// TwinCAT 3 PLC project FTP
// ProgramVersion: 3.1.4023.0
// libraries:
//   Tc2_FTP, * (Beckhoff Automation GmbH)
//   Tc2_Standard, * (Beckhoff Automation GmbH)
//   Tc2_System, * (Beckhoff Automation GmbH)
//   Tc3_Module, * (Beckhoff Automation GmbH)
// project tree:
//   / GlobalTextList.TcGTLO, PlcTask.TcTTO, Visualization Manager.TcVMO (not stored)
//   POUs/ MAIN.TcPOU
//   VISUs/ FTP.TcVIS
// real-time tasks:
//   TASK PlcTask: cycle T#10ms, priority 20, ADS port 350
//   TASK PlcTask1: cycle T#10ms, priority 21, ADS port 351
//   TASK PlcTask2: cycle T#10ms, priority 22, ADS port 352
//   TASK PlcTask3: cycle T#10ms, priority 23, ADS port 353
//   TASK PlcTask4: cycle T#10ms, priority 24, ADS port 354
//   TASK PlcTask5: cycle T#10ms, priority 25, ADS port 355
//   TASK PlcTask6: cycle T#10ms, priority 26, ADS port 356

CONFIGURATION FTP
    RESOURCE PLC ON TwinCAT3
        TASK PlcTask(INTERVAL := T#10ms, PRIORITY := 20);
        PROGRAM MAIN WITH PlcTask : MAIN;
    END_RESOURCE
END_CONFIGURATION

// ---- POUs/MAIN.TcPOU
PROGRAM MAIN

VAR_INPUT
END_VAR

VAR_OUTPUT
	progressBar: UDINT;
END_VAR

VAR
	FB_FTP_FileUploadEx: FB_FTP_FileUploadEx;
END_VAR

FB_FTP_FileUploadEx(
			sHost:= 'ftp.dlptest.com',
			nPort:= 21, 
			sUsername:= 'dlpuser@dlptest.com',
			sPassword:= 'SzMf7rTE4pCrf9dV286GuNe4N',
			sSrcFile:= 'C:\Users\Kasper\Desktop\JensIsJens.txt', 
			sDesFile:= 'Casper2.csv', 
			bExecute:= TRUE, 
			tTimeout:= T#15S, 
			bBusy=> , 
			bError=> , 
			nErrId=> , 
			nProgress=> progressBar);

END_PROGRAM

// ---- GlobalTextList.TcGTLO
TEXTLIST GlobalTextList
  581 = 'SYNC'
  221 = 'UPLOAD'
END_TEXTLIST

// ---- VISUs/FTP.TcVIS
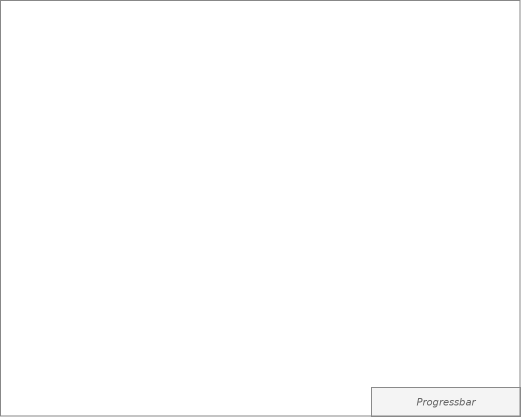
VISUALIZATION FTP  // 521x417
    Progressbar (371,387 150x30), variable: MAIN.progressBar
END_VISUALIZATION
